FUNCTION_BLOCK ABSTRACT FB_AxisControl EXTENDS FB_BaseAxis IMPLEMENTS I_Axis
VAR_INPUT
	bMoveAxis				: BOOL;		// Move azimuth to given position
	bTracking				: BOOL;		// enable tracking
	bStopAxis				: BOOL;		// stop the Axis
	fMinPosition			: REAL := 0;
	fMaxPosition			: REAL := 450.0;
	fCalibPosition			: LREAL := 45.0; // // current position of the calibration cam
END_VAR
VAR_OUTPUT
END_VAR
VAR
	fSlewTime				: LREAL;	// time to reach target position

	InDigitalInputs	  AT%I*	: WORD;		// digitale inputs der Endlagen
	InDiagnostic	  AT%I*	: UDINT;	// diagnostic number
	InTorque	 	  AT%I*	: INT;		// derotator torque feedback
	IbSTO		  	  AT%I*	: BOOL;		// STO

	fbAxisCalibration		: MC_SetPosition;

	axisEvent			: FB_EventLog;
	diagnosticEvent		: FB_EventLog;
	
	bDiagnosticError		: BOOL;
	
	fbReadParameter		: MC_ReadParameter;
	bGetLastPosition		: BOOL := TRUE;
	
	calibrationEvent		: FB_Eventlog;
	fTorque			: REAL;	// percentage of the derotator torque
	torqueWarning			: FB_EventLog;	
END_VAR
VAR PERSISTENT
	fLastPosition			: LREAL := -1.0;
END_VAR

PROPERTY isTracking : BOOL
GET
isTracking := fbAxis.isTracking;
END_GET
END_PROPERTY

PROPERTY MoveAxis : BOOL
GET
MoveAxis := bMoveAxis;
END_GET
SET
bMoveAxis := MoveAxis;
END_SET
END_PROPERTY

PROPERTY MoveDone : BOOL
GET
MoveDone := fbAxis.MoveDone;
END_GET
END_PROPERTY

PROPERTY SlewTime : LREAL
GET
SlewTime := fSlewTime;
END_GET
END_PROPERTY

PROPERTY StopAxis : BOOL
GET
StopAxis := bStopAxis;
END_GET
SET
bStopAxis := StopAxis;
END_SET
END_PROPERTY

PROPERTY Tracking : BOOL
GET
Tracking := bTracking;
END_GET
SET
bTracking := Tracking;
END_SET
END_PROPERTY

END_FUNCTION_BLOCK

(* stored: Version 1.1.0.1, ProductVersion 3.1.4024.15
   POU FB_AxisControl: Id {6fdef2a3-176a-42ec-90be-24250bb425eb}, SpecialFunc None
   Property isTracking: Id {d14d4ed7-aa44-40b8-a06b-dbd9bb4bc398}
   Get Get: Id {d8cce5f4-c21e-4d9a-87e8-69b1f87cb648}
   Property MoveAxis: Id {62370465-c9c4-4b3d-9522-670fc80fcf7d}
   Get Get: Id {b6a037c9-1a5a-4ccc-a67e-cd8fbf875616}
   Set Set: Id {d5ee563e-2fbb-4a6b-ae57-cdb88f0e5477}
   Property MoveDone: Id {ffed8cc8-8f25-4253-859b-58a4e017102a}
   Get Get: Id {9b084521-bbd8-4f17-b07f-9acdda778b7d}
   Property SlewTime: Id {a36dc70d-226a-4ef7-9e23-e0fd5a5024cb}
   Get Get: Id {87871d10-1142-4737-afba-11d3d9c70605}
   Property StopAxis: Id {895eb35b-1f81-42b7-8416-fc32b401fd0f}
   Get Get: Id {d8fe8d4f-84fc-4959-900d-984362d0d694}
   Set Set: Id {7b322eb7-7271-44c8-a7b2-c7ee70ff43dc}
   Property Tracking: Id {4bf1bf93-5980-423d-96c9-58edc9fdb938}
   Get Get: Id {e9371fc2-0020-4b0a-85b6-17721f14dcf3}
   Set Set: Id {4ff2f8a4-67a6-4244-b8ba-f5f82d04fc0f} *)
